FUNCTION Matrix_ElementProduct : BOOL
VAR_INPUT
	A : REFERENCE TO Matrix;
	B : REFERENCE TO Matrix;
	Res : REFERENCE TO Matrix;
END_VAR
VAR
	I : UINT;
END_VAR

IF NOT(A.IsEqualSize(Res)) OR A.IsEmpty THEN
	Matrix_ElementProduct := FALSE;
	RETURN;
END_IF

IF NOT(B.IsEqualSize(Res)) OR B.IsEmpty THEN
	Matrix_ElementProduct := FALSE;
	RETURN;
END_IF

Matrix_ElementProduct := TRUE;

FOR I := 0 TO Res.Length - 1 DO
	Res.SetI(I,A.GetI(I)*B.GetI(I));
END_FOR

END_FUNCTION

(* stored: Version 1.1.0.1, ProductVersion 3.1.4024.9
   POU Matrix_ElementProduct: Id {61941b80-cefc-03b0-068a-f4ffeccad5f5}, SpecialFunc None *)
